TYPE ST_LOG_WriteImageData :
STRUCT
	aLogPT			: ARRAY[0..65000] OF BYTE;
	aLogML			: ARRAY[0..65000] OF BYTE;
	aLogOT			: ARRAY[0..65000] OF BYTE;
	aLogCT			: ARRAY[0..65000] OF BYTE;
END_STRUCT
END_TYPE

(* stored: Version 1.1.0.1
   DUT ST_LOG_WriteImageData: Id {afdbf980-d7f3-48d2-93ed-ab477fa5324b} *)
